/// Axis move relative parameter strucure
TYPE ST_AxisMoveRelParameter EXTENDS ST_AxisMoveParameter :
STRUCT
	/// Distance
	fDistance: LREAL;
END_STRUCT
END_TYPE

(* stored: Version 1.1.0.1, ProductVersion 3.1.4022.9
   DUT ST_AxisMoveRelParameter: Id {ca18a397-d96c-42ff-bd6b-4bce392e8b5d} *)
